FUNCTION_BLOCK RfidHead EXTENDS TcoCore.TcoComponent
VAR_OUTPUT

END_VAR
VAR
    _itfRfidHeadWrapper : IRfidHeadWrapper;
    _readUidTask        : ReadUidTask(THIS^);
    _readDataTask       : ReadDataTask(THIS^);
    _writeDataTask      : WriteDataTask(THIS^);
    _lockTask           : LockTask(THIS^);
    _resetTask          : ResetTaskRfid(THIS^);

    _rfidInOut      : RfidInOut;
    _errorId        : RFID_FB_U.ERROR;
    _uiDataRxLength : UINT;

END_VAR

Map();

_readUidTask(rfidInOut := _rfidInOut, ActionDesc := '<#ReadUid#>');
_readDataTask(rfidInOut := _rfidInOut, ActionDesc := '<#ReadData#>');
_writeDataTask(rfidInOut := _rfidInOut, ActionDesc := '<#WriteData#>');
_lockTask(rfidInOut := _rfidInOut, ActionDesc := '<#WriteData#>');
_resetTask(rfidInOut := _rfidInOut, ActionDesc := '<#ResetTask#>');

PROPERTY Data : Tc2_System.T_MaxString
GET
Data := _readDataTask.Data;
END_GET
END_PROPERTY

PROPERTY DataRxLength : UINT
GET
DataRxLength := _uiDataRxLength;
END_GET
END_PROPERTY

{attribute 'monitoring' := 'call'}
PROPERTY ErrorId : RFID_FB_U.ERROR
GET
{warning disable C0371}
ErrorId := _readDataTask.ErrorId or _readUidTask.ErrorId or _writeDataTask.ErrorId OR _lockTask.ErrorId;
END_GET
END_PROPERTY

METHOD FB_init : BOOL
VAR_INPUT
    bInitRetains       : BOOL; // if TRUE, the retain variables are initialized (warm start / cold start)
    bInCopyCode        : BOOL; // if TRUE, the instance afterwards gets moved into the copy code (online change)
    ParentObject       : ITcoObject;
    itfRfidHeadWrapper : IRfidHeadWrapper;
    udiTimeOut         : TIME;
END_VAR
VAR
    _microToMillis : UDINT := 1000;
END_VAR
// This is not clear to me... I from time to time the consumer code does not see 'FB_init' of 'TcoObject', that's why overridden here with super call...
{warning disable C0316}
SUPER^.FB_init(bInitRetains, bInCopyCode, ParentObject);

THIS^._itfRfidHeadWrapper := itfRfidHeadWrapper;

THIS^._rfidInOut.udiTimeOut := TIME_TO_UDINT(udiTimeOut) * _microToMillis;

_readUidTask.FB_init
(
    bInitRetains   := bInitRetains
    , bInCopyCode  := bInCopyCode
    , ParentObject := ParentObject
);
END_METHOD

{attribute 'monitoring' := 'call'}
PROPERTY IsError : BOOL
GET
//collected Error from Tasks
IsError :=
    this^.pReadUidTask.Error or this^.pReadDataTask.Error or this^.pLockTask.Error or this^.pWriteDataTask.Error;
END_GET
END_PROPERTY

METHOD LockMethod : TcoCore.ITcoTaskStatus
VAR_INPUT
    udiDataLength : UINT;  //Length of the Data to read
    StartAdress   : UDINT; // Memory Adress, from which to start
END_VAR
IF (pLockTask <> 0) THEN
    _rfidInOut.uiDataLenght   := udiDataLength;
    _rfidInOut.udiStartAdress := StartAdress;
    LockMethod                := pLockTask.Invoke();
END_IF
END_METHOD

METHOD Private Map : BOOL
_itfRfidHeadWrapper.Execute
(
    xExecute              := _rfidInOut.xExecute
    , xAbort              := _rfidInOut.xAbort
    , udiTimeOut          := _rfidInOut.udiTimeOut
    , eCommand            := _rfidInOut.eCommand
    , udiStartAdress      := _rfidInOut.udiStartAdress
    , uiDataLenght        := _rfidInOut.uiDataLenght
    , myWriteData         := _rfidInOut.myWriteData
    , myReadData          => _rfidInOut.myReadData
    , xDone               => _rfidInOut.xDone
    , xBusy               => _rfidInOut.xBusy
    , xError              => _rfidInOut.xError
    , xAborted            => _rfidInOut.xAborted
    , eErrorID            => _rfidInOut.eErrorID
    , xTP                 => _rfidInOut.xTP
    , xRWHeadNotCOnnected => _rfidInOut.xRWHeadNotCOnnected
    , uiDataRxLength      => _rfidInOut.uiDataRxLength
);
END_METHOD

PROPERTY pLockTask : TcoCore.ITcoTask
GET
pLockTask := _lockTask;
END_GET
END_PROPERTY

PROPERTY pReadDataTask : TcoCore.ITcoTask
GET
pReadDataTask := _readDataTask;
END_GET
END_PROPERTY

PROPERTY pReadUidTask : TcoCore.ITcoTask
GET
pReadUidTask := _readUidTask;
END_GET
END_PROPERTY

PROPERTY pResetTask : TcoCore.ITcoTask
GET
pResetTask := _resetTask;
END_GET
END_PROPERTY

PROPERTY pWriteDataTask : TcoCore.ITcoTask
GET
pWriteDataTask := _writeDataTask;
END_GET
END_PROPERTY

METHOD ReadDataMethod : TcoCore.ITcoTaskStatus
VAR_INPUT
    udiDataLength : UINT; //Length of the Data to read
    MemoryAddr    : BYTE; // Memory Adress, from which to start
END_VAR
IF (pReadDataTask <> 0) THEN
    _rfidInOut.uiDataLenght   := udiDataLength;
    _rfidInOut.udiStartAdress := MemoryAddr;
    _uiDataRxLength           := _rfidInOut.uiDataRxLength;
    ReadDataMethod            := pReadDataTask.Invoke();
END_IF
END_METHOD

METHOD ReadUidMethod : TcoCore.ITcoTaskStatus
VAR_INPUT
END_VAR
IF (pReadUidTask <> 0) THEN
    ReadUidMethod := pReadUidTask.Invoke();
END_IF
END_METHOD

METHOD ResetMethod : TcoCore.ITcoTaskStatus
IF (pResetTask <> 0) THEN
    ResetMethod := pResetTask.Invoke();
END_IF
END_METHOD

(*~
    <docu>
        <summary>
            Restore all tasks of this instance into initial state.
        </summary>
    </docu>
~*)
METHOD Restore : ITcoRestorable

IF (pReadUidTask <> 0) THEN
    pReadUidTask.Restore();
END_IF;

IF (pReadDataTask <> 0) THEN
    pReadDataTask.Restore();
END_IF;

IF (pWriteDataTask) <> 0 THEN
    pWriteDataTask.Restore();
END_IF

IF (pLockTask) <> 0 THEN
    pLockTask.Restore();
END_IF

IF (pResetTask) <> 0 THEN
    pResetTask.Restore();
END_IF
END_METHOD

METHOD PROTECTED ServiceMode
END_METHOD

PROPERTY Uid : Tc2_System.T_MaxString
GET
Uid := _readUidTask.Uid;
END_GET
END_PROPERTY

METHOD WriteDataMethod : TcoCore.ITcoTaskStatus
VAR_IN_OUT
    WriteData : ARRAY[*] OF BYTE; //Data to write to Tag
END_VAR
VAR_INPUT
    MemoryAddr : BYTE; // Memory Adress, from which to start
END_VAR
VAR_INST
    _i : DINT;
END_VAR
IF (pWriteDataTask <> 0) THEN
    _rfidInOut.uiDataLenght   := SIZEOF(WriteData);
    _rfidInOut.udiStartAdress := MemoryAddr;

    FOR _i := LOWER_BOUND(WriteData, 1) TO UPPER_BOUND(WriteData, 1) DO
        _rfidInOut.myWriteData[_i] := WriteData[_i];
    END_FOR

    _uiDataRxLength := _rfidInOut.uiDataRxLength;
    WriteDataMethod := pWriteDataTask.Invoke();
END_IF
END_METHOD

END_FUNCTION_BLOCK

(* stored: Version 1.1.0.1, ProductVersion 3.1.4024.12
   POU RfidHead: Id {b9804aa8-9ded-4408-aa6f-fd33a940430f}, SpecialFunc None
   Folder Map: Id {3dfaf2b8-ee21-4439-afca-07a7d42a308e}
   Folder Operations: Id {df559028-2e02-4963-aa18-db1bf643b042}
   Folder Output: Id {fadfd011-b785-4463-ad2e-7e9e2fbad96c}
   Folder Status: Id {cdd118b6-d89c-4268-9c74-33451fb6a01f}
   Folder Tasks: Id {d35bf5df-58c3-4edc-bf2e-00dbc08d63df}
   Property Data: Id {1fb1a294-0f74-49b6-aca2-ef87b4d04c1b}
   Get Get: Id {0b8ab245-d033-4aa1-8c3b-3fa6bfeccb26}
   Property DataRxLength: Id {70d6b81e-2898-4615-a665-a92937e07bee}
   Get Get: Id {acd058f0-6fbf-469a-848a-48f46330c28a}
   Property ErrorId: Id {35979862-d9a0-4a81-9c0f-e464d21ecf76}
   Get Get: Id {ab9af534-dbda-476d-9287-e93a1b84bb40}
   Method FB_init: Id {acc83f3d-a253-476c-ba4c-e2ba4ba3fab2}
   Property IsError: Id {d9d3a25a-cbe3-47a2-b502-99367ed0072f}
   Get Get: Id {dee70cac-df4b-4d91-a940-519204f87392}
   Method LockMethod: Id {5b8af782-9258-483b-9db7-a2ba2851c196}
   Method Map: Id {ff22a4d1-e2da-4e1f-915e-50fba519f1cc}
   Property pLockTask: Id {ed95084c-9316-4d1b-9d7f-77e04b21bd90}
   Get Get: Id {804f4cee-15df-41ea-8b76-8e3b38f36ac1}
   Property pReadDataTask: Id {021e5c43-cbf7-42ab-bed9-348ea02c82b2}
   Get Get: Id {f9657344-727f-468c-94f0-a9392f36803f}
   Property pReadUidTask: Id {75d0b3bb-dad0-46cc-b9ce-c4fe8da6c1a1}
   Get Get: Id {a4eea792-fc9d-4933-bed5-6171c33d92b8}
   Property pResetTask: Id {b296bb90-d596-4976-bf8b-1db2b7483cbf}
   Get Get: Id {5d74eafc-aa46-4077-8d5f-1d19773ffd83}
   Property pWriteDataTask: Id {51d3690b-728e-43b4-bd8e-60414670f7b3}
   Get Get: Id {7ad9dcca-5d4b-43dd-9182-f8ead9f44ab3}
   Method ReadDataMethod: Id {3aee4692-ee7a-4a0f-8d95-4524ec406de7}
   Method ReadUidMethod: Id {0635c5a9-1d48-4c5b-9edb-aa7456a44eb8}
   Method ResetMethod: Id {abbada54-6015-4715-9323-328dc5d2a08d}
   Method Restore: Id {60e8ad41-0936-485d-81f4-a441c90de548}
   Method ServiceMode: Id {d3fef0af-a61e-4c69-9748-134dd26773e4}
   Property Uid: Id {6d4473c0-eb64-4022-8d44-8853c97ae5f9}
   Get Get: Id {9e4f55a5-1e9c-40d8-9ab9-7c808c7c075a}
   Method WriteDataMethod: Id {e9cf36cf-4bbd-4615-8f53-70f3a520d6f9} *)
